FUNCTION F_ChargePointStatusToString : STRING(31)
VAR_INPUT
	eStatus : E_OCPP1_ChargePointStatus;
END_VAR

CASE eStatus OF
	E_OCPP1_ChargePointStatus.Available: F_ChargePointStatusToString := 'Available';
	E_OCPP1_ChargePointStatus.Preparing: F_ChargePointStatusToString := 'Preparing';
	E_OCPP1_ChargePointStatus.Charging: F_ChargePointStatusToString := 'Charging';
	E_OCPP1_ChargePointStatus.SuspendedEVSE: F_ChargePointStatusToString := 'SuspendedEVSE';
	E_OCPP1_ChargePointStatus.SuspendedEV: F_ChargePointStatusToString := 'SuspendedEV';
	E_OCPP1_ChargePointStatus.Finishing: F_ChargePointStatusToString := 'Finishing';
	E_OCPP1_ChargePointStatus.Reserved: F_ChargePointStatusToString := 'Reserved';
	E_OCPP1_ChargePointStatus.Unavailable: F_ChargePointStatusToString := 'Unavailable';
	E_OCPP1_ChargePointStatus.Faulted: F_ChargePointStatusToString := 'Faulted';
END_CASE

END_FUNCTION

(* stored: Version 1.1.0.1
   POU F_ChargePointStatusToString: Id {01f142c5-1a8a-4010-a5bb-66664228919d}, SpecialFunc None *)
